FUNCTION_BLOCK FB_Extends EXTENDS FB_Base
VAR_INPUT
    bStart : BOOL;
END_VAR

END_FUNCTION_BLOCK

(* stored: Version 1.1.0.1
   POU FB_Extends: Id {11111111-1111-1111-1111-111111111102} *)
